# EPICS substitutions: iocs/simulationTest/simulationTestApp/Db/simulation_test.substitutions
# EtherCAT Master

file $(ETHERCAT)/db/MASTER.template
{
pattern {       DEVICE , PORT    , SCAN     }
        { rjq35657:sim , MASTER0 , "I/O Intr" }
}

#
# EL1014:
# 4 channel 24V digital input
#
file $(ETHERCAT)/db/EL1014.template
{
pattern {  DEVICE     , PORT   , SCAN     }
        { rjq35657:M1 , DIGIN0 , "I/O Intr" }
}
